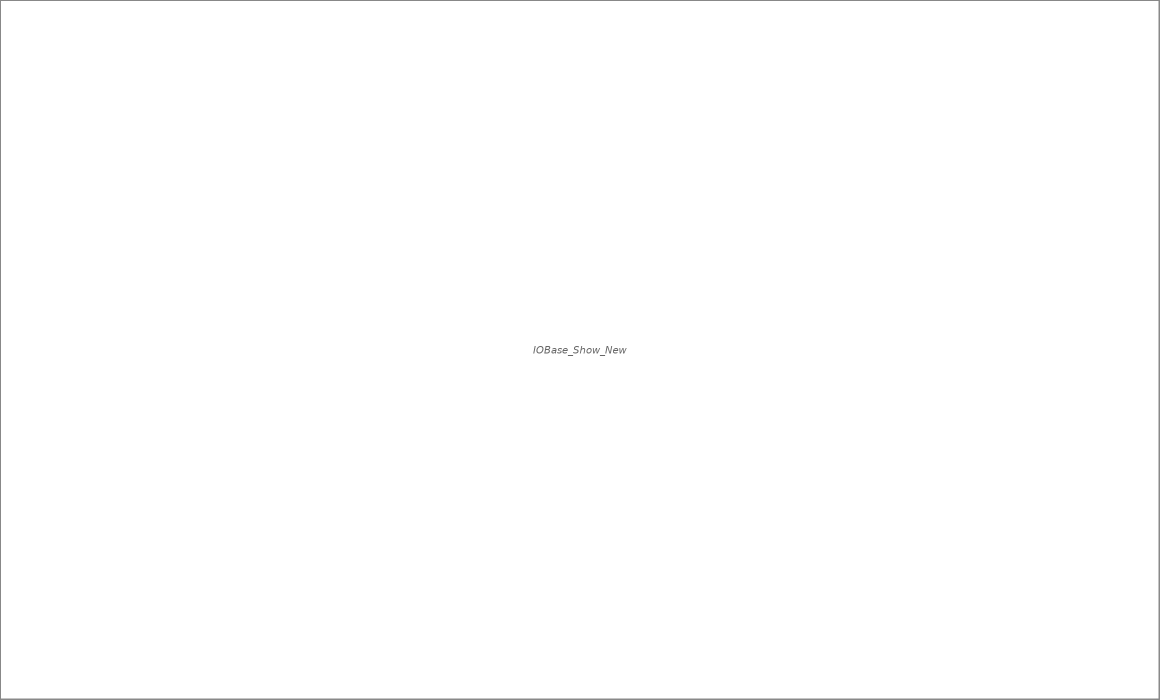
VISUALIZATION IO_Input  // 1160x700
    TabControl (0,0 1160x700)
        shows IOBase_Show_New(userData := TesterIO.fbIOBase_Input.HMIITF)
        [0]: TabTitle=Input
END_VISUALIZATION

(* stored: Version 1.1.0.1, ProductVersion 3.1.4024.4
   Visu IO_Input: Id {0e88059a-09f8-4b96-8f7d-885cd0e0a7a2} *)
